{attribute 'qualified_only'}
{attribute 'strict'}
{attribute 'to_string'}
TYPE MotionStatus :
(
	ConstantVelocity,
	Accelerating,
	Decelerating
);
END_TYPE

(* stored: Version 1.1.0.1, ProductVersion 3.1.4026.18
   DUT MotionStatus: Id {0a6dc904-10d7-093f-3ac7-a0f7a91569a8} *)
